// TIA Portal V19 export
VAR_GLOBAL   // PLC tag table "Test"
   test1 AT %M120.0 : Bool;
   test2 AT %M120.1 : Bool;
END_VAR
